FUNCTION CheckDivReal : REAL
VAR_INPUT
	divisor: REAL;
END_VAR
VAR_EXTERNAL
	fbCheckDivRealInfo: FB_CheckDivRealInfo;
END_VAR

(*This function checks if a division by zero is performed*)

fbCheckDivRealInfo(
	rDivisor			:= divisor,
	sLogMessage	=> ,
	rReturnDivReal 	=> CheckDivReal);

END_FUNCTION

(* stored: Version 1.1.0.1, ProductVersion 3.1.4024.12
   POU CheckDivReal: Id {9d80fe98-c4af-4f3b-a271-d21c68372537}, SpecialFunc CheckDivReal32 *)
